FUNCTION Convert_SINT_TO_USINT : Hresult
VAR_INPUT
	in : SINT;
	out : REFERENCE TO USINT;
END_VAR
VAR
	converted : USINT;
END_VAR

converted := SINT_TO_USINT(in);

IF (USINT_TO_SINT(converted) <> in) THEN
	Convert_SINT_TO_USINT := INCOMPATIBLE;
	RETURN;
END_IF

out := converted;

END_FUNCTION

(* stored: Version 1.1.0.1, ProductVersion 3.1.4024.12
   POU Convert_SINT_TO_USINT: Id {cb8a1a34-912b-4588-9423-0531711f0ff1}, SpecialFunc None *)
